INTERFACE I_StringLookupElement EXTENDS I_Fallible


METHOD LookupAtomicMass : LREAL
VAR_INPUT
    sLookup : STRING;
END_VAR
END_METHOD


METHOD LookupAtomicNumber : INT
VAR_INPUT
    sLookup : STRING;
END_VAR
END_METHOD


METHOD LookupDensity : LREAL
VAR_INPUT
    sLookup : STRING;
END_VAR
END_METHOD

END_INTERFACE

(* stored: Version 1.1.0.1
   Itf I_StringLookupElement: Id {ba7a2c21-deb3-474b-b7eb-995f7adb6478}
   Method LookupAtomicMass: Id {913d3b19-2087-41aa-8e5c-39fc748f1444}
   Method LookupAtomicNumber: Id {5f83cf7a-fc59-42db-9ede-3a362b64e71d}
   Method LookupDensity: Id {3579ce78-6b57-4a66-ad8f-4e83b829e31d} *)
